Fanuc KAREL source: CNV_JPOS_REL.kl

PROGRAM T
%NOLOCKGROUP
VAR
 v0 : JOINTPOS
 v1 : ARRAY[9] OF REAL
 v2 : INTEGER
BEGIN
 CNV_JPOS_REL(v0, v1, v2)
END T
